// Mitsubishi GX Works2 project: Hil   PLC: FX2N/FX2NC

// global labels: Global1
VAR_GLOBAL
  Verdiendring_1 : Verdiendring;
  Settpunkt_Kp_glob AT D2 : REAL;
  Settpunkt_Ki_glob AT D4 : REAL;
  Settpunkt_Kd_glob AT D6 : REAL;
  Settpunkt_Referanse_glob AT D0 : INT;
  Tf_glob AT D8 : REAL;
  Tankp AT D10 : REAL;
  fP_glob AT D12 : REAL;
  fI_glob AT D14 : REAL;
  fDD AT D16 : REAL;
  Referanse_glob : INT;
  Kp_glob : REAL;
  Ki_glob : REAL;
  Kd_glob : REAL;
  Pådrag AT D20 : REAL;
  PID_REGULATOR_1 : PID_REGULATOR;
END_VAR

// task Task_01 (event TRUE, interval 0, priority 31): POU_01

PROGRAM POU_01
(* structured ladder/FBD written out as ST: instructions are called as NAME(EN, inputs, outputs); _pN, _eN, _tN stand for wires *)
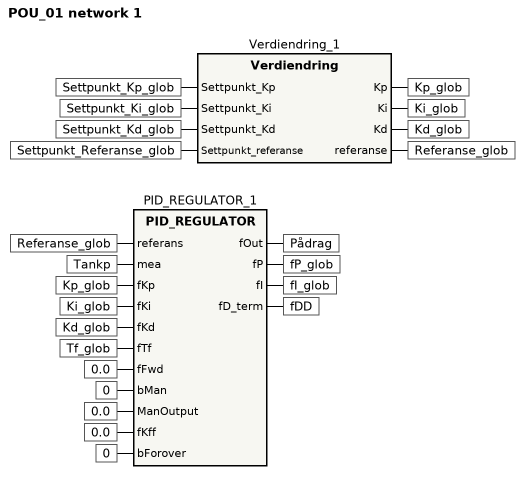
(* network 1 *)
Verdiendring_1(Settpunkt_Kp := Settpunkt_Kp_glob, Settpunkt_Ki := Settpunkt_Ki_glob, Settpunkt_Kd := Settpunkt_Kd_glob, Settpunkt_referanse := Settpunkt_Referanse_glob, Kp => Kp_glob, Ki => Ki_glob, Kd => Kd_glob, referanse => Referanse_glob);
PID_REGULATOR_1(referans := Referanse_glob, mea := Tankp, fKp := Kp_glob, fKi := Ki_glob, fKd := Kd_glob, fTf := Tf_glob, fFwd := 0.0, bMan := 0, ManOutput := 0.0, fKff := 0.0, bForover := 0, fOut => Pådrag, fP => fP_glob, fI => fI_glob, fD_term => fDD);
END_PROGRAM

FUNCTION_BLOCK PID_REGULATOR
VAR_INPUT
  referans : INT;
  mea : REAL;
  fKp : REAL;
  fKi : REAL;
  fKd : REAL;
END_VAR
VAR_OUTPUT
  fOut : REAL;
  fP : REAL;
END_VAR
VAR
  fError : REAL;
END_VAR
VAR_OUTPUT
  fI : REAL;
END_VAR
VAR CONSTANT
  fTi : REAL := 10;
END_VAR
VAR
  fTs : REAL;
END_VAR
VAR_OUTPUT
  fD_term : REAL;
END_VAR
VAR
  fError_prev : REAL;
  fTracking : REAL;
END_VAR
VAR CONSTANT
  fNom : REAL := 4.0;
END_VAR
VAR
  bUseI : BOOL;
  bUseD : BOOL;
END_VAR
VAR_INPUT
  fTf : REAL;
END_VAR
VAR CONSTANT
  fTd : REAL := 1.0;
END_VAR
VAR
  fDfilter : REAL;
  fRawOut : REAL;
END_VAR
VAR_INPUT
  fFwd : REAL;
END_VAR
VAR
  bUseFwd : BOOL;
END_VAR
VAR_INPUT
  bMan : BOOL;
END_VAR
VAR
  fRef : REAL;
  fKt : REAL;
  fManOutput : REAL;
END_VAR
VAR CONSTANT
  fOutMax : REAL := 100.0;
END_VAR
VAR
  bSaturated : BOOL;
END_VAR
VAR CONSTANT
  fOutMin : REAL;
  input : BOOL := TRUE;
END_VAR
VAR_INPUT
  ManOutput : REAL;
  fKff : REAL;
  bForover : BOOL;
END_VAR
VAR
  bUseI_prev : BOOL;
  skan : INT;
  fskan : REAL;
  bInit : BOOL;
END_VAR
FLT(input,referans,fRef);

MOV(TRUE, D8010, skan);
FLT(TRUE, skan, fskan);
fTs := fskan/10000.0;

(* Initialiser I-ledd på første syklus til steady-state *)
  IF bInit THEN
      fI      := fNom;
      fDfilter := 0.0;
      bInit   := FALSE;
  END_IF;

bUseI := fKi > 0.0;
bUseD := fKd > 0.0;

fError:= fRef - mea;

(* P-ledd *)
fP:= fKp*fError;

(* I-ledd *)
IF bUseI THEN

        fI := fI + fTs * (fKi * fError + fTracking);

ELSE
    fI := fNom;
END_IF;
bUseI_prev := bUseI;

(* D-ledd *)
IF bUseD AND fTf > 0.0 THEN
    fDfilter := fDfilter + fTs / fTf * (fKd / fTs * (fError - fError_prev) - fDfilter);
    fD_term := fDfilter;
ELSE
    fD_term := 0.0;
END_IF;

(* foroverkobling *)
fRawOut := fP + fI + fD_term;
IF bForover THEN
    fRawOut := fRawOut + (fFwd * fKff);
END_IF;


IF bMan THEN
    fOut := ManOutput;
    (* Tracking: hold I-ledd oppdatert = rykkfri overgang til auto *)
    fI   := ManOutput - fP- fD_term;
ELSE
    (* Begrens output *)
    IF fRawOut > fOutMax THEN
        fOut    := fOutMax;
        bSaturated := TRUE;
    ELSIF fRawOut < fOutMin THEN
        fOut    := fOutMin;
        bSaturated := TRUE;
    ELSE
        fOut    := fRawOut;
        bSaturated := FALSE;
    END_IF;

    (* Anti-windup tracking signal *)
    fKt := fKi / fKp; (* 1/Ti *)
    fTracking := fKt * (fOut - fRawOut);
END_IF;

 fError_prev:=fError;
END_FUNCTION_BLOCK

FUNCTION_BLOCK Verdiendring
VAR
  Rampe_1 : Rampe;
END_VAR
VAR_INPUT
  Settpunkt_Kp : REAL;
  Settpunkt_Ki : REAL;
  Settpunkt_Kd : REAL;
END_VAR
VAR_OUTPUT
  Kp : REAL;
  Ki : REAL;
  Kd : REAL;
  referanse : INT;
END_VAR
VAR_INPUT
  Settpunkt_referanse : INT;
END_VAR
VAR
  fSettpunkt_referanse : REAL;
  fReferanse : REAL;
  Rampe_2 : Rampe;
  Rampe_3 : Rampe;
  Rampe_4 : Rampe;
  iRateSek : INT;
END_VAR
(* structured ladder/FBD written out as ST: instructions are called as NAME(EN, inputs, outputs); _pN, _eN, _tN stand for wires *)
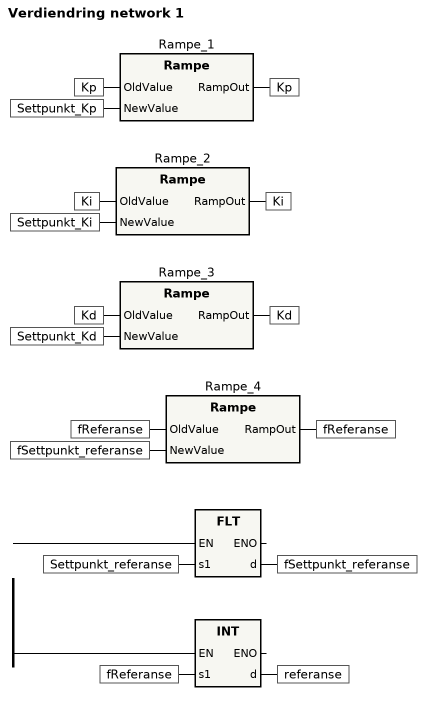
(* network 1 *)
Rampe_1(OldValue := Kp, NewValue := Settpunkt_Kp, RampOut => Kp);
Rampe_2(OldValue := Ki, NewValue := Settpunkt_Ki, RampOut => Ki);
Rampe_3(OldValue := Kd, NewValue := Settpunkt_Kd, RampOut => Kd);
Rampe_4(OldValue := fReferanse, NewValue := fSettpunkt_referanse, RampOut => fReferanse);
FLT(TRUE, Settpunkt_referanse, fSettpunkt_referanse);
INT(TRUE, fReferanse, referanse);
END_FUNCTION_BLOCK

FUNCTION_BLOCK Rampe
VAR_INPUT
  OldValue : REAL;
  NewValue : REAL;
END_VAR
VAR
  RampStep : REAL;
END_VAR
VAR_OUTPUT
  RampOut : REAL;
END_VAR
VAR
  rStartValue : REAL;
  rProgress : REAL;
  rLastTarget : REAL;
  rT_smooth : REAL;
END_VAR
VAR CONSTANT
  fRateSek : REAL := 5.0;
END_VAR


IF fRateSek > 0.0 THEN
	RampStep := 1.0 / (fRateSek * 100.0);
END_IF;

IF NewValue <> rLastTarget THEN
    rStartValue  := RampOut;
    rProgress    := 0.0;
    rLastTarget  := NewValue;
END_IF;

IF rProgress < 1.0 THEN
    rProgress := rProgress + RampStep;

    IF rProgress > 1.0 THEN
        rProgress := 1.0;
    END_IF;

    (*Smoothstep funksjon, formel: 3t² - 2t³ *)	
    rT_smooth := rProgress * rProgress * (3.0 - (2.0 * rProgress));

    RampOut := rStartValue + ((NewValue - rStartValue) * rT_smooth);
ELSE
    RampOut := NewValue;
END_IF;
END_FUNCTION_BLOCK
